TYPE HandlingComRequest :
STRUCT
  Start : BOOL;
  Stop : BOOL;
  GoHome : BOOL;
  Halt : BOOL;
END_STRUCT
END_TYPE

(* stored: Version 1.1.0.1
   DUT HandlingComRequest: Id {739baffe-f4ca-4f4b-ab35-6591eb51762a} *)
